FUNCTION Convert_LWORD_TO_LINT : BOOL
VAR_INPUT
	in : LWORD;
	out : REFERENCE TO LINT;
END_VAR
VAR
	converted : LINT;
END_VAR

converted := LWORD_TO_LINT(in);

IF (LINT_TO_LWORD(converted) <> in) THEN
	RETURN;
END_IF

out := converted;
Convert_LWORD_TO_LINT := TRUE;

END_FUNCTION

(* stored: Version 1.1.0.1, ProductVersion 3.1.4024.12
   POU Convert_LWORD_TO_LINT: Id {85eb80d6-c347-4c3e-9968-a837874cd9f5}, SpecialFunc None *)
